FUNCTION_BLOCK Robot
VAR_OUTPUT
	forceStop AT %Q* : BOOL;
	resetSignal AT %Q* : BOOL;
	
	outputs AT %Q* : ARRAY[1..50] OF INT;
	inputs AT %I* : ARRAY[1..20] OF INT;
	
	taskID : INT;
	
	completedTask : INT;
	tool : SectionEnum;
	
	operational : BOOL;
	reserved : BOOL;
	reservation : SectionEnum := SectionEnum.NULL_SECTION;
	
	ready : BOOL;
	done : BOOL;
	error : BOOL;
	errId : DINT;
END_VAR
VAR
	step : (SEND_COMMAND, WAIT);
END_VAR

taskID := outputs[1];

completedTask := inputs[1];

IF completedTask = taskID THEN
	done := TRUE;
END_IF

METHOD command : BOOL
VAR_INPUT
	task : INT;
	param1 : INT;
	param2 : INT;
	param3 : INT;
END_VAR
//command := reserve();

//IF command THEN
	(*
	taskId := task;
	parameters[1] := param1;
	parameters[2] := param2;
	parameters[3] := param3;
	*)
	
	outputs[1] := task;
	outputs[2] := param1;
	outputs[3] := param2;
	outputs[4] := param3;
//END_IF
END_METHOD

METHOD commandEx : BOOL
VAR_INPUT
	newOutputs : REFERENCE TO ARRAY[1..50] OF INT;
END_VAR
outputs := newOutputs;
END_METHOD

METHOD eStop : BOOL
VAR_INPUT
END_VAR
forceStop := TRUE;
eStop := TRUE;
END_METHOD

METHOD release : BOOL
VAR_INPUT
	sectionReservation : SectionEnum;
END_VAR
IF reservation = sectionReservation AND reserved THEN
	reservation := -1;
	reserved := FALSE;
	release := TRUE;
END_IF
END_METHOD

METHOD reserve : BOOL
VAR_INPUT
	sectionReservation : SectionEnum;
END_VAR
(*
this method exists because chipboard and wood bunk operations use the same robot
both sections need to check if the robot is open to commands before use
*)
IF
	(reserved AND reservation = SectionReservation) OR_ELSE
	(NOT reserved OR sectionReservation = SectionEnum.NULL_SECTION)
THEN
	reservation := sectionReservation;
	reserved := TRUE;
	reserve := TRUE;
END_IF
END_METHOD

METHOD reset : BOOL
//resetSignal := TRUE;
//done := FALSE;

MEMSET(ADR(outputs), 0, SIZEOF(outputs));
(*
IF ready AND completedTask = 0 THEN
	resetSignal := FALSE;
	reset := TRUE;
END_IF
*)
END_METHOD

METHOD resume : BOOL
VAR_INPUT
END_VAR
forceStop := FALSE;

resume := NOT error AND errId = 0;
END_METHOD

METHOD setCommandAndWait : BOOL
VAR_INPUT
	newOutputs : REFERENCE TO ARRAY[1..50] OF INT;
END_VAR
outputs := newOutputs;

IF done THEN
	(*	
	IF NOT reset() THEN
		RETURN;
	END_IF
	
	step := 0;
	*)
	setCommandAndWait := TRUE;
END_IF
END_METHOD

END_FUNCTION_BLOCK

(* stored: Version 1.1.0.1, ProductVersion 3.1.4024.11
   POU Robot: Id {870b17d8-8fed-45ea-b532-f3f727b3e8ec}, SpecialFunc None
   Folder Obsolete: Id {866be447-1963-4a08-8cb7-28bb42cb4605}
   Method command: Id {6180ebeb-6fb3-4e45-8d5f-010642c60433}
   Method commandEx: Id {55c20752-492d-4e9a-a647-f2d920916f43}
   Method eStop: Id {974b2363-087f-4f71-a37b-fdee6dacfa65}
   Method release: Id {7fed4361-8a94-445d-8040-f071f846d639}
   Method reserve: Id {1e01deef-588d-4739-a104-23ce337539cb}
   Method reset: Id {89eb6678-027f-45a1-a94f-ae23b58ecc5c}
   Method resume: Id {1d12dfe1-c8ff-4b57-9b31-0d4b08a72b4a}
   Method setCommandAndWait: Id {861e79f4-9d73-4326-81bf-3ad217fcca64} *)
